Staubli VAL3: Queue.dtx

public num nPush
public num nPop
public num nElems
public MotionCmd buffer[10]
  [0]
    mdesc mDesc = {leave=0, reach=0}
    num nDuration
    num nSequence
    joint jJoint
  [1]
    mdesc mDesc = {leave=0, reach=0}
    num nDuration
    num nSequence
    joint jJoint
  [2]
    mdesc mDesc = {leave=0, reach=0}
    num nDuration
    num nSequence
    joint jJoint
  [3]
    mdesc mDesc = {leave=0, reach=0}
    num nDuration
    num nSequence
    joint jJoint
  [4]
    mdesc mDesc = {leave=0, reach=0}
    num nDuration
    num nSequence
    joint jJoint
  [5]
    mdesc mDesc = {leave=0, reach=0}
    num nDuration
    num nSequence
    joint jJoint
  [6]
    mdesc mDesc = {leave=0, reach=0}
    num nDuration
    num nSequence
    joint jJoint
  [7]
    mdesc mDesc = {leave=0, reach=0}
    num nDuration
    num nSequence
    joint jJoint
  [8]
    mdesc mDesc = {leave=0, reach=0}
    num nDuration
    num nSequence
    joint jJoint
  [9]
    mdesc mDesc = {leave=0, reach=0}
    num nDuration
    num nSequence
    joint jJoint
